{attribute 'linkalways'} 
{attribute 'no_explicit_call' := 'This FB is a CLASS and must be accessed using methods or properties'}
{attribute 'enable_dynamic_creation'}
FUNCTION_BLOCK Node_F_VN_FlipImage EXTENDS VisionNode
VAR
	ipSrcImage : _ITcVnImage;
    ipDestImage : _ITcVnImage;
    eFlipAxis : _ETcVnFlipAxis(ETcVnFlipAxis.TCVN_FA_X);
    hrPrev : _HRESULT(S_OK);
	hresult : _HRESULT(S_OK);
END_VAR

METHOD PUBLIC  Clone : I_Node
VAR
	pNode : POINTER TO Node_F_VN_FlipImage;
END_VAR
pNode := __NEW(Node_F_VN_FlipImage);
Clone := pNode^;
END_METHOD

METHOD FB_init : BOOL
VAR_INPUT
	bInitRetains : BOOL; // if TRUE, the retain variables are initialized (warm start / cold start)
	bInCopyCode : BOOL;  // if TRUE, the instance afterwards gets moved into the copy code (online change)
END_VAR
AddInput('ipSrcImage', ipSrcImage);
AddInput('hrPrev', hrPrev);
AddOutput('ipDestImage', ipDestImage);
AddOutput('hresult',hresult);
AddParameter('eFlipAxis', eFlipAxis);
END_METHOD

METHOD PROTECTED  OnExecute : HRESULT
hresult.Value := F_VN_FlipImage(
	ipSrcImage := ipSrcImage.Value, 
	ipDestImage := ipDestImage.Value, 
	eFlipAxis := eFlipAxis.Value, 
	hrPrev := hrPrev.Value);
END_METHOD

METHOD PUBLIC PreExecutionCheck
VAR_INPUT
	Check : I_PreExecutionChecks;
END_VAR
IF FAILED(hrPrev.Value) THEN
    RETURN;
END_IF

Check.IsTrue(ipSrcImage.IsValid, 'ipSrcImage must contain an image');
END_METHOD

END_FUNCTION_BLOCK

(* stored: Version 1.1.0.1, ProductVersion 3.1.4024.13
   POU Node_F_VN_FlipImage: Id {a6f99e12-a793-04fc-29f7-a3f276999bb5}, SpecialFunc None
   Folder Constructor: Id {be4bcdf3-492d-03c4-3f42-dba786bbac7e}
   Method Clone: Id {dfef732d-7cc2-0902-2f27-11a30313b0e4}
   Method FB_init: Id {4d071b0a-447c-07fd-16c1-9fa35ffa874e}
   Method OnExecute: Id {07193c4d-c45e-07df-3cec-b934b2aefaf5}
   Method PreExecutionCheck: Id {5869bb14-d849-097b-3049-e3ca8572dcb4} *)
